PROGRAM FUKUDA_MOVE
//FUNCTION FUKUDA_MOVE : BOOL
VAR_INPUT
	STEP_DATA_1: BYTE;
	STEP_DATA_2: BYTE;
	STEP_DATA_3: BYTE;
	STEP_DATA_4: BYTE;
	STEP_DATA_5: BYTE;
	FUKUDA_HOME: INT;
END_VAR

VAR
	
	(*
	DataWordInput1 AT %IB100 : ARRAY [0..15] OF WORD; 
	DataWordInput2 AT %IB132 : ARRAY [16..31] OF WORD; 
	DataWordInput3 AT %IB164 : ARRAY [32..47] OF WORD; 
	DataWordInput4 AT %IB196 : ARRAY [48..56] OF WORD; 
	DataWordOutput1 AT %QB100 : ARRAY [0..15] OF WORD; 
	DataWordOutput2 AT %QB132 : ARRAY [16..31] OF WORD; 
	DataWordOutput3 AT %QB164 : ARRAY [32..47] OF WORD; 
	DataWordOutput4 AT %QB196 : ARRAY [48..56] OF WORD; 
	*)
	Gateway_Q0_MODE_COMMAND_0 AT %QX100.0 : BOOL ;
	Gateway_Q0_MODE_COMMAND_1 AT %QX100.1 : BOOL ;
	Gateway_Q0_RESET AT %QX100.4 : BOOL;
	Gateway_Q0_RESTART AT %QX100.5 : BOOL;
	Gateway_Q0_STOP AT %QX100.7 : BOOL;
	Gateway_Q1_0 AT %QX101.0 : BOOL;
	Gateway_Q1_1 AT %QX101.1 : BOOL;
	Gateway_Q1_2 AT %QX101.2 : BOOL;
	Gateway_Q1_3 AT %QX101.3 : BOOL;
	Gateway_Q1_4 AT %QX101.4 : BOOL;
	Gateway_Gateway_Unit_2_Status AT %QB102 : BYTE;
	Gateway_Q3_0 AT %QX103.0 : BOOL;
	Gateway_Q3_1 AT %QX103.1 : BOOL;
	Gateway_Q3_2 AT %QX103.2 : BOOL;
	Gateway_Q3_3 AT %QX103.3 : BOOL;	
	

	ID1_StepData AT %QB114 : BYTE;
	ID1_Hold AT %QX115.0 : BOOL;
	ID1_SVON AT %QX115.1 : BOOL;
	ID1_Drive AT %QX115.2 : BOOL;
	ID1_Reset AT %QX115.3 : BOOL;
	ID1_Setup AT %QX115.4 : BOOL;
	

	ID2_StepData AT %QB134 : BYTE;
	ID2_Hold AT %QX135.0 : BOOL;
	ID2_SVON AT %QX135.1 : BOOL;
	ID2_Drive AT %QX135.2 : BOOL;
	ID2_Reset AT %QX135.3 : BOOL;
	ID2_Setup AT %QX135.4 : BOOL;


	ID3_StepData AT %QB154 : BYTE;
	ID3_Hold AT %QX155.0 : BOOL;
	ID3_SVON AT %QX155.1 : BOOL;
	ID3_Drive AT %QX155.2 : BOOL;
	ID3_Reset AT %QX155.3 : BOOL;
	ID3_Setup AT %QX155.4 : BOOL;
	
	
	ID4_StepData AT %QB174 : BYTE;
	ID4_Hold AT %QX175.0 : BOOL;
	ID4_SVON AT %QX175.1 : BOOL;
	ID4_Drive AT %QX175.2 : BOOL;
	ID4_Reset AT %QX175.3 : BOOL;
	ID4_Setup AT %QX175.4 : BOOL;
	

	ID5_StepData AT %QB194 : BYTE;
	ID5_Hold AT %QX195.0 : BOOL;
	ID5_SVON AT %QX195.1 : BOOL;
	ID5_Drive AT %QX195.2 : BOOL;
	ID5_Reset AT %QX195.3 : BOOL;
	ID5_Setup AT %QX195.4 : BOOL;
	
	byte0 : BYTE;
	byte1 : BYTE;
	byte2 : BYTE;
	byte3 : BYTE;
	
	bit14_0 : BOOL;
	bit14_1 : BOOL;
	bit14_2 : BOOL;
	bit14_3 : BOOL;
	bit14_4 : BOOL;
	bit14_5 : BOOL;
	
	bit15_0 : BOOL;
	bit15_1 : BOOL;
	bit15_2 : BOOL;
	bit15_3 : BOOL;
	bit15_4 : BOOL; 
	
	bit34_0 : BOOL;
	bit34_1 : BOOL;
	bit34_2 : BOOL;
	bit34_3 : BOOL;
	bit34_4 : BOOL;
	bit34_5 : BOOL;
	
	bit35_0 : BOOL;
	bit35_1 : BOOL;
	bit35_2 : BOOL;
	bit35_3 : BOOL;
	bit35_4 : BOOL; 
	
	bit54_0 : BOOL;
	bit54_1 : BOOL;
	bit54_2 : BOOL;
	bit54_3 : BOOL;
	bit54_4 : BOOL;
	bit54_5 : BOOL;
	
	bit55_0 : BOOL;
	bit55_1 : BOOL;
	bit55_2 : BOOL;
	bit55_3 : BOOL;
	bit55_4 : BOOL; 
	
	bit74_0 : BOOL;
	bit74_1 : BOOL;
	bit74_2 : BOOL;
	bit74_3 : BOOL;
	bit74_4 : BOOL;
	bit74_5 : BOOL;
	
	bit75_0 : BOOL;
	bit75_1 : BOOL;
	bit75_2 : BOOL;
	bit75_3 : BOOL;
	bit75_4 : BOOL; 
	
	bit94_0 : BOOL;
	bit94_1 : BOOL;
	bit94_2 : BOOL;
	bit94_3 : BOOL;
	bit94_4 : BOOL;
	bit94_5 : BOOL;
	
	bit95_0 : BOOL;
	bit95_1 : BOOL;
	bit95_2 : BOOL;
	bit95_3 : BOOL;
	bit95_4 : BOOL; 	
	
	ID1_I0_MODE_COMMAND_0 AT %IX100.0 : BOOL :=0;
	ID1_I0_MODE_COMMAND_1 AT %IX100.1 : BOOL:=0;
	ID1_I0_READY AT %IX100.4 : BOOL;
	ID1_I0_ALARM AT %IX100.5 : BOOL;
	ID1_I0_INITIAL AT %IX100.6 : BOOL;
	ID1_I0_COMMUNICATING AT %IX100.7 : BOOL;
	ID1_I1_0 AT %IX101.0 : BOOL;
	ID1_I1_1 AT %IX101.1 : BOOL;
	ID1_I1_2 AT %IX101.2 : BOOL;
	ID1_I1_3 AT %IX101.3 : BOOL;
	ID1_I1_4 AT %IX101.4 : BOOL;
	ID1_I2_0 AT %IX102.0 : BOOL;
	ID1_I2_1 AT %IX102.1 : BOOL;
	ID1_I2_2 AT %IX102.2 : BOOL;
	ID1_I2_3 AT %IX102.3 : BOOL;
	ID1_I2_4 AT %IX102.4 : BOOL;

	ID1_I3_0 AT %IX103.0 : BOOL;
	ID1_I3_1 AT %IX103.1 : BOOL;
	
	ID1_I32_0 AT %IX132.0 : BOOL;
	ID1_I32_1 AT %IX132.1 : BOOL;
	ID1_I33_0 AT %IX133.0 : BOOL;
	ID1_I33_1 AT %IX133.1 : BOOL;
(*-----------------------------------------------------------*)

	iTest15: SINT;
	iTest16: SINT;
	
	bTest1 : BOOL;
	bTest2 : BOOL;
	bTest3 : BOOL;
	bTest4 : BOOL;
	bTest5 : BOOL;
	bTest6 : BOOL;
	bTest7 : BOOL;
	bTest8 : BOOL;
	bTest9 : BOOL;
	bTest10 : BOOL;
	bTest11 : BOOL;
	bTest12 : BOOL;
	bTest13 : BOOL;
	bTest14 : BOOL;
	
	StepData1 : BYTE;
	StepData2 : BYTE;
	StepData3 : BYTE;
	StepData4 : BYTE;
	StepData5 : BYTE;
	
	star :BOOL;
	hom : BOOL;

	reset: BOOL;
	
	ID1_ALARM AT%IX115.7 : BOOL;
	ID2_ALARM AT%IX135.7 : BOOL;
	ID3_ALARM AT%IX155.7 : BOOL;
	ID4_ALARM AT%IX175.7 : BOOL;
	ID5_ALARM AT%IX195.7 : BOOL;
	
	ID1_SVRE AT%IX115.1 : BOOL;
	ID2_SVRE AT%IX135.1 : BOOL;
	ID3_SVRE AT%IX155.1 : BOOL;
	ID4_SVRE AT%IX175.1 : BOOL;
	ID5_SVRE AT%IX195.1 : BOOL;
	
	ID1_INP AT%IX115.3 : BOOL;
	ID2_INP AT%IX135.3 : BOOL;
	ID3_INP AT%IX155.3 : BOOL;
	ID4_INP AT%IX175.3 : BOOL;
	ID5_INP AT%IX195.3 : BOOL;
	
	PROSES: STRING;
	STAGE: INT;
	
	PROCESS: INT;
	START_PROCESS: BOOL;
	STEP_DATAS: INT;
	PROCESS_DELAY: TIME :=T#300MS;
	FUKUDA_RUNNING: BOOL :=FALSE;
	ACTIVE_STEPDATA : BYTE;
	//ACTIVE_ID: INT :=1;
	TMR1: TON;
	TMR2: TON;
	TMR3: TON;
	TMR4: TON;
	TMR5: TON;
	TMR6: TON;
	TMR10: Ton;
	TMR11: TON;
	TMR12: TON;
	TMR13: TON;
	TMR14: TON;
	TMR20: TON;
	TMR21: TON;
	TMR22: TON;
	TMR23: TON;
	TMR30: TON;
	TMR31: TON;
	TMR32: TON;
	TMR33: TON;
	TMR40: TON;
	TMR41: TON;
	TMR42: TON;
	TMR43: TON;
	TMR50: TON;
	TMR51: TON;
	TMR52: TON;
	TMR53: TON;
	
	
	TMR101: TON;
	TMR102: TON;
	TMR103: TON;
	TMR104: TON;
	TMR105: TON;
	TMR106: TON;
	ID5: INT;
	TMR7: Ton;
	TMR_RES_CARTSN: TOF;
	TMR_ACTIVATE_RESET: TON;
END_VAR


PROCESS_DELAY:= T#400MS;
IF 	INPUT_VAR.ACTIVE_ID >=0 THEN
STEP_DATA_1:=STEP_DATA_1+1;

IF STEP_DATA_2>=5 THEN
	STEP_DATA_2:=STEP_DATA_2+1;
END_IF

STEP_DATA_3:=STEP_DATA_3+1;	
END_IF


IF NOT INPUT_VAR.FUKUDA_HOME THEN //fukuda_running THEN
	IF  ID1_SVRE AND ID2_SVRE  AND  ID3_SVRE AND  ID4_SVRE AND  ID5_SVRE THEN
		TMR1(IN:=TRUE,PT:=T#0.5S);
		TMR4(IN:=TRUE,PT:=T#3S);
		TMR5(IN:=TRUE,PT:=T#3.5S);
		TMR6(IN:=TRUE,PT:=T#25S);
		IF ID1_SVRE THEN
			ID1_SETUP :=TMR5.Q;
		ELSE
			ID1_SVON :=TRUE;	
		END_IF

		IF ID2_SVRE THEN
			ID2_SETUP :=TMR1.Q;
		ELSE
			ID2_SVON :=TRUE;	
		END_IF
	
		IF ID3_SVRE THEN
		ID3_SETUP :=TMR4.Q;
		ELSE
			ID3_SVON :=TRUE;	
		END_IF
		CASE INPUT_VAR.I_CURRENT_TRANSACTION.TRANSPORT_INDEX OF
		1:
			TMR2(IN:=TRUE,PT:=T#1S);
			IF ID4_SVRE THEN
				ID4_SETUP :=TMR2.Q;
			ELSE
				ID4_SVON :=TRUE;	
			END_IF
		2:
			TMR3(IN:=TRUE,PT:=T#1.5S);
			IF ID5_SVRE THEN
				ID5_SETUP :=TMR3.Q;
			ELSE
				ID5_SVON :=TRUE;	
			END_IF
		END_CASE

	//IF TMR6.Q THEN
	IF ID1_INP AND ID2_INP AND ID3_INP AND (ID4_INP OR ID5_INP) THEN
		ID1_SETUP :=FALSE;
		ID2_SETUP :=FALSE;
		ID3_SETUP :=FALSE;
		ID4_SETUP :=FALSE;
		ID5_SETUP :=FALSE;
	
		TMR1(IN:=FALSE);
		TMR2(IN:=FALSE);
		TMR3(IN:=FALSE);
		TMR4(IN:=FALSE);
		TMR5(IN:=FALSE);
	//ACTIVE_ID:=1;
	//FUKUDA_RUNNING:=TRUE;
		INPUT_VAR.FUKUDA_HOME:=TRUE;
	END_IF
	
	ELSE
				
	ID1_SVON :=TRUE;
	ID2_SVON :=TRUE;
	ID3_SVON :=TRUE;
	ID4_SVON :=TRUE;
	ID5_SVON :=TRUE;

	END_IF
ELSE
	TMR6(IN:=FALSE);

	CASE INPUT_VAR.ACTIVE_ID OF
	0:
		INPUT_VAR.I_CASE:=INPUT_VAR.I_CASE+1;
		//INPUT_VAR.I_FUKUDA_RUNNING:=FALSE;
		INPUT_VAR.ACTIVE_ID:=6;
		
	1:
		IF STEP_DATA_1 = 0 THEN
			INPUT_VAR.ACTIVE_ID:=2;
		ELSE
			IF ID1_ALARM THEN
				Reset := TRUE;
				TMR10(IN:=TRUE,PT:= PROCESS_DELAY);
				IF TMR10.Q THEN
					Reset := FALSE;
				END_IF
			ELSE
				ID1_StepData :=STEP_DATA_1;
				ID1_Drive := FALSE;
				TMR11(IN:=TRUE,PT:= PROCESS_DELAY);
				IF TMR11.Q THEN
					IF ID1_INP THEN
					ID1_Drive := TRUE;
					TMR12(IN:=TMR11.Q,PT:= PROCESS_DELAY);
					IF TMR12.Q THEN
						ID1_Drive := FALSE;
						INPUT_VAR.ACTIVE_ID:=2;
						TMR10(IN:=FALSE);
						TMR11(IN:=FALSE);
						TMR12(IN:=FALSE);
						INPUT_VAR.FUKUDA_HOME:=TRUE;
					END_IF
					END_IF
				END_IF
			END_IF
		END_IF
	//	INPUT_VAR.I_CASE:=INPUT_VAR.I_CASE+1;
		//INPUT_VAR.I_FUKUDA_RUNNING:=FALSE;
	2:
		IF STEP_DATA_2 = 0 THEN
			INPUT_VAR.ACTIVE_ID:=3;
		ELSE
			
			IF ID2_ALARM THEN
				Reset := TRUE;
				TMR20(IN:=TRUE,PT:= PROCESS_DELAY);
				IF TMR20.Q THEN
					Reset := FALSE;
				END_IF
			ELSE
			ID2_StepData :=STEP_DATA_2;
			TMR21(IN:=TRUE,PT:= PROCESS_DELAY);
			IF TMR21.Q THEN
				ID2_Drive := TRUE;
				TMR22(IN:=TMR21.Q,PT:= PROCESS_DELAY);
				IF TMR22.Q THEN
				IF ID2_INP THEN
					ID2_Drive := FALSE;
					INPUT_VAR.ACTIVE_ID:=3;
					TMR20(IN:=FALSE);
					TMR21(IN:=FALSE);
					TMR22(IN:=FALSE);
				END_IF
				END_IF
			END_IF
			END_IF
		END_IF
	3:
		IF STEP_DATA_3 = 0 THEN
			INPUT_VAR.ACTIVE_ID:=4;
		ELSE
			
		IF ID3_ALARM THEN
			Reset := TRUE;
			TMR30(IN:=START_PROCESS,PT:= PROCESS_DELAY);
			IF TMR30.Q THEN
				Reset := FALSE;
			END_IF
		ELSE
		
		ID3_StepData :=STEP_DATA_3;
		TMR31(IN:=TRUE,PT:= PROCESS_DELAY);
		IF TMR31.Q THEN
			ID3_DRIVE := TRUE;	
			TMR32(IN:=TMR31.Q,PT:= PROCESS_DELAY);
			
			IF TMR32.Q THEN
				IF  ID3_INP THEN
				ID3_Drive := FALSE;
				INPUT_VAR.ACTIVE_ID:=4;
				TMR30(IN:=FALSE);
				TMR31(IN:=FALSE);
				TMR32(IN:=FALSE);
				END_IF
			END_IF
		END_IF
		END_IF
	END_IF
4:
		IF STEP_DATA_4 = 0 THEN
			INPUT_VAR.ACTIVE_ID:=5;
		ELSE
			IF ID4_ALARM THEN
				Reset := TRUE;
				TMR40(IN:=TRUE,PT:= PROCESS_DELAY);
				IF TMR40.Q THEN
					Reset := FALSE;
				END_IF
			ELSE
			
			ID4_StepData :=STEP_DATA_4;
			TMR41(IN:=TRUE,PT:= PROCESS_DELAY);
			IF TMR41.Q THEN
				ID4_Drive := TRUE;
				TMR42(IN:=TMR41.Q,PT:= PROCESS_DELAY);
				
				IF TMR42.Q THEN
					ID4_Drive := FALSE;
					INPUT_VAR.ACTIVE_ID:=5;
					TMR40(IN:=FALSE);
					TMR41(IN:=FALSE);
					TMR42(IN:=FALSE);
				END_IF
			END_IF
			END_IF
		END_IF
	5:
		IF STEP_DATA_5 = 0 THEN
			INPUT_VAR.ACTIVE_ID:=0;
		ELSE
			
			IF ID5_ALARM THEN
				Reset := TRUE;
				TMR50(IN:=TRUE,PT:= PROCESS_DELAY);
				IF TMR50.Q THEN
					Reset := FALSE;
				END_IF
			ELSE
			
			ID5_StepData :=STEP_DATA_5;
			TMR51(IN:=TRUE,PT:= PROCESS_DELAY);
			IF TMR51.Q THEN
				ID5_Drive := TRUE;	
				TMR52(IN:=TMR51.Q,PT:= PROCESS_DELAY);
				IF TMR52.Q THEN
					ID5_Drive := FALSE;
					INPUT_VAR.ACTIVE_ID:=0;
					TMR50(IN:=FALSE);
					TMR51(IN:=FALSE);
					TMR52(IN:=FALSE);
			
				END_IF
			END_IF
			END_IF
		END_IF
		
END_CASE 

	//START_PROCESS := FALSE;
END_IF
TMR7(IN:=reset,PT:= T#1S);
IF  tmr7.Q THEN
	reset:=FALSE;
END_IF
IF ID1_ALARM OR ID2_ALARM OR ID3_ALARM OR ID4_ALARM OR ID5_ALARM THEN
			reset:=TRUE;
			ELSE
				reset:=FALSE;
			END_IF
IF reset THEN
	ID1_Reset := TRUE;
	ID2_Reset := TRUE;
	ID3_Reset := TRUE;
	ID4_Reset := TRUE;
	ID5_Reset := TRUE;
	TMR_ACTIVATE_RESET(IN:=TRUE,PT:=T#10S);
	IF TMR_ACTIVATE_RESET.Q THEN
		TMR_RES_CARTSN(IN:=TRUE,PT:=T#0.5S);
	END_IF
	
ELSE
	TMR_ACTIVATE_RESET(IN:=FALSE);
	TMR_RES_CARTSN(IN:=FALSE);
	ID1_Reset := FALSE;
	ID2_Reset := FALSE;
	ID3_Reset := FALSE;
	ID4_Reset := FALSE;
	ID5_Reset := FALSE;
END_IF
INPUT_VAR.O_RESET_CARTESSIAN := TMR_RES_CARTSN.Q;

END_PROGRAM

(* stored: Version 1.1.0.1, ProductVersion 3.1.4020.12
   POU FUKUDA_MOVE: Id {a9aa7c17-a8da-4255-b975-1708592af896}, SpecialFunc None *)
